KUKA KRL program: ItemPick.src, ItemPick.dat

--- ItemPick.src ---
&ACCESS RVP
&PARAM EDITMASK = *
DEF ItemPick()
   ; ItemPickExample
   ; --------------
   ; Demonstrates bin-picking using roboception's ItemPick module with continuous detection
   ; and pick-and-place operations.
   ;
   ; The program:
   ; 1. Continuously detects items in a bin using vision system
   ; 2. For each detected item, attempts multiple grasp poses if needed
   ; 3. Places successfully picked items at a predefined location
   ; 4. Loops until no more items are detected or program is interrupted
   ;
   ; ENHANCEMENTS:
   ; - Clean 3-tier speed hierarchy (High/Medium/Slow) for easy configuration
   ; - Collision detection support with gripper ID and pre-grasp offsets
   ; - Proper separation of movement offsets vs. detection offsets
   ; - Consistent use of .dat file variables for better maintainability
   ;

   ; Parameters for detection - declared in .dat file
   DECL INT CURRENTITEM, IT

   ; Service name - same as the EKI service name
   ; TODO: Change this to the correct service name - could be "sensor_a_pipeline_1_rc_itempick-compute_grasps"
   serviceNameDetect[] = "rc_itempick-compute_grasps"

   ; Maximum number of grasps to process per detection
   MAX_GRASPS_TO_PROCESS = 1
   ; Maximum number of detection retries
   MAX_DETECTION_RETRIES = 5

   ; Detection parameters
   SUCTION_LENGTH = 0.09  ; Updated to match EKI specification
   SUCTION_WIDTH = 0.02   ; Matches EKI specification
   ITEM_TYPE[] = "BAG"  ; "BAG" for bags or " " for any other item
   LOAD_CARRIER_ID[] = " " ; Single space to represent empty/none
   ROI_ID[] = "roi_bags"
   POSE_FRAME[] = "external"

   ; Collision detection parameters - use " " to skip sending
   GRIPPER_ID[] = "SingleVacuum"    ; Gripper identifier for collision detection
   DET_PRE_GRASP_X_OFFSET = 0.0     ; Detection pre-grasp offset in X direction (m) - SEPARATE from movement offset
   DET_PRE_GRASP_Y_OFFSET = 0.0     ; Detection pre-grasp offset in Y direction (m) - SEPARATE from movement offset
   DET_PRE_GRASP_Z_OFFSET = -0.1    ; Detection pre-grasp offset in Z direction (m) - SEPARATE from movement offset

   ; Gripping parameters
   PRE_GRASP_Z_OFFSET = -100   ; in 100 mm above (along item frame z)
   PRE_PLACE_Z_OFFSET = -100   ; in mm (along world z)

   ; NOTE: Movement uses PRE_GRASP_Z_OFFSET, detection uses DET_PRE_GRASP_Z_OFFSET
   ; These are two different parameters that can be configured independently!

   ;FOLD INI;%{PE}
      ;FOLD BASISTECH INI
         GLOBAL INTERRUPT DECL 3 WHEN $STOPMESS==TRUE DO IR_STOPM ( )
         INTERRUPT ON 3
         BAS (#INITMOV,0 )
      ;ENDFOLD (BASISTECH INI)
   ;ENDFOLD (INI)

   INTERRUPT DECL 89 WHEN $flag[998] DO RC_NOTIFYRECEIVED(1, 998)
   INTERRUPT ON 89

   ;FOLD SPTP home vel=75 % HIGH Speed Transit ;%{pe}
      SPTP XHOME WITH $VEL_AXIS[1] = SVEL_JOINT(ptpSpeedHigh)
   ;ENDFOLD

   GRIPPERBLOW()

   RC_INIT(serviceNameDetect[])

   ;
   ; Main program loop
   ; Continuously tries to detect and pick items until no more items are found
   ; or the program is interrupted
   ;
   LOOP
      RC_SETMSG("Detect next item.")

      ;
      ; Detection retry loop
      ; Attempts to detect items up to MAX_DETECTION_RETRIES times
      ; Exits either on successful detection or when max retries are reached
      ;
      FOR IT = 1 TO MAX_DETECTION_RETRIES
         ; Configure detection parameters using helper function
         ; Sets up item type, pose frame, load carrier, ROI, suction surface, and collision detection parameters
         RC_CONFIGUREPARAMS(serviceNameDetect[], ITEM_TYPE[], POSE_FRAME[], LOAD_CARRIER_ID[], ROI_ID[], SUCTION_LENGTH, SUCTION_WIDTH, GRIPPER_ID[], DET_PRE_GRASP_X_OFFSET, DET_PRE_GRASP_Y_OFFSET, DET_PRE_GRASP_Z_OFFSET)

         ; Perform detection
         ; Sends detection request to vision system and waits for response
         PerformDetection(serviceNameDetect[])

         ; Exit retry loop if detection was successful
         IF DetectionSuccessful() THEN
            EXIT
         ENDIF

         ; Exit program if we've exhausted all retries
         IF IT == MAX_DETECTION_RETRIES THEN
            RC_SETMSG("No more items detected - ending program")
            EXIT
         ENDIF
      ENDFOR

      ;
      ; Process detected grasps
      ; If detection was successful, attempt to pick and place each detected grasp
      ; If detection failed, exit the program
      ;
      IF DetectionSuccessful() THEN
         ; Process grasps from this detection, up to MAX_GRASPS_TO_PROCESS
         FOR CURRENTITEM = 1 TO NUMDETECTEDGRASPS
            GRASP = DETECTEDGRASPS[CURRENTITEM]
            LogGraspInfo(CURRENTITEM, GRASP)
            ExecutePickAndPlace(GRASP, PLACEPOSE, PRE_GRASP_Z_OFFSET, PRE_PLACE_Z_OFFSET)

            ; Break if we've processed maximum number of grasps
            IF CURRENTITEM >= MAX_GRASPS_TO_PROCESS THEN
               EXIT
            ENDIF
         ENDFOR
      ELSE
         ; No items detected after all retries - exit program
         EXIT
      ENDIF
   ENDLOOP

   ; Clean up and return home

   ;FOLD SPTP home vel=75 % HIGH Speed Transit ;%{pe}
      SPTP XHOME WITH $VEL_AXIS[1] = SVEL_JOINT(ptpSpeedHigh)
   ;ENDFOLD
END

DEF ExecutePickAndPlace(GRASPPOSE:IN, PLACEPOSE:IN, PRE_GRASP_Z_OFFSET:IN, PRE_PLACE_Z_OFFSET:IN)
   ;
   ; Executes a complete pick and place operation
   ;
   ; @param GRASPPOSE: Target pose for grasping the object
   ; @param PLACEPOSE: Target pose for placing the object
   ; @param PRE_GRASP_Z_OFFSET: Vertical offset (mm) for pre-grasp approach position
   ; @param PRE_PLACE_Z_OFFSET: Vertical offset (mm) for pre-place approach position
   ; @return TRUE if operation successful, FALSE if vacuum check fails
   ;
   DECL FRAME GRASPPOSE
   DECL E6POS PLACEPOSE
   DECL REAL PRE_GRASP_Z_OFFSET, PRE_PLACE_Z_OFFSET

   ; Internal pose calculations
   DECL FRAME PREGRASPPOSE, PREPLACEPOSE
   DECL FRAME F_OFFSET

   ; Calculate pre-grasp pose
   F_OFFSET = $NULLFRAME
   F_OFFSET.Z = PRE_GRASP_Z_OFFSET
   PREGRASPPOSE = GRASPPOSE:F_OFFSET

   ; Calculate pre-place pose
   PREPLACEPOSE.x = PLACEPOSE.x
   PREPLACEPOSE.y = PLACEPOSE.y
   PREPLACEPOSE.z = PLACEPOSE.z - PRE_PLACE_Z_OFFSET
   PREPLACEPOSE.a = PLACEPOSE.a
   PREPLACEPOSE.b = PLACEPOSE.b
   PREPLACEPOSE.c = PLACEPOSE.c

   ; Move over bin - HIGH speed transit
   SPTP OVERBINPOSE WITH $VEL_AXIS[1] = SVEL_JOINT(ptpSpeedHigh)

   ; Move to pre-grasp - MEDIUM speed approach
   SLIN PREGRASPPOSE with $vel = svel_cp(linSpeedMedium, , lDatMedium), $tool = stool2(fDatDefault), $base = sbase(fDatDefault.base_no)

   ; Move to grasp - SLOW speed for careful in-bin movement
   SLIN GRASPPOSE with $vel = svel_cp(linSpeedSlow, , lDatSlow), $tool = stool2(fDatDefault), $base = sbase(fDatDefault.base_no)

   RC_SETMSG("Grasp position reached. Suctioning...")
   GRIPPERSUCK()

   ; Exit bin - SLOW speed for careful movement out of bin
   SLIN PREGRASPPOSE with $vel = svel_cp(linSpeedSlow, , lDatSlow), $tool = stool2(fDatDefault), $base = sbase(fDatDefault.base_no)

   IF GripperHasVacuumIO THEN
      ; Execute place sequence - HIGH speed transit to place area
      SPTP PREPLACEPOSE with $vel_axis[1] = svel_joint(ptpSpeedHigh), $tool = stool2(fDatDefault), $base = sbase(fDatDefault.base_no), $ipo_mode = sipo_mode(fDatDefault.ipo_frame), $load = sload(fDatDefault.tool_no), $acc_axis[1] = sacc_joint(pDatHigh), $apo = SAPO_PTP(pDatHigh), $gear_jerk[1] = sgear_jerk(pDatHigh), $collmon_tol_pro[1] = use_cm_pro_values(0)
      ; Place item - MEDIUM speed for controlled placement
      SLIN PLACEPOSE with $vel = svel_cp(linSpeedMedium, , lDatMedium), $tool = stool2(fDatDefault), $base = sbase(fDatDefault.base_no)
      GRIPPERBLOW()
      ; Return from place - HIGH speed transit movement
      SPTP PREPLACEPOSE with $vel_axis[1] = svel_joint(ptpSpeedHigh), $tool = stool2(fDatDefault), $base = sbase(fDatDefault.base_no), $ipo_mode = sipo_mode(fDatDefault.ipo_frame), $load = sload(fDatDefault.tool_no), $acc_axis[1] = sacc_joint(pDatHigh), $apo = SAPO_PTP(pDatHigh), $gear_jerk[1] = sgear_jerk(pDatHigh), $collmon_tol_pro[1] = use_cm_pro_values(0)
   ELSE
      RC_SETMSG("No vacuum - moving on...")
      GRIPPERBLOW()
   ENDIF
END

; ---- Helper Functions ----
;FOLD GRIPPERSUCK
   DEF GRIPPERSUCK()
      WAIT SEC 0.0
      GripperBlowIO = false
      GripperSuckIO = true
      WAIT SEC 1.0
   END
;ENDFOLD (GRIPPERSUCK)

;FOLD GRIPPERBLOW
   DEF GRIPPERBLOW()
      WAIT SEC 0.0
      GripperBlowIO = true
      GripperSuckIO = false
   END
;ENDFOLD (GRIPPERSUCK)

; ---- Roboception Functions ----
;FOLD ROBOCEPTION_FUNCTIONS
   ;FOLD RC_CONFIGUREPARAMS
      DEF RC_CONFIGUREPARAMS(serviceNameDetect[]:IN, ITEM_TYPE[]:IN, POSE_FRAME[]:IN, LOAD_CARRIER_ID[]:IN, ROI_ID[]:IN, SUCTION_LENGTH:IN, SUCTION_WIDTH:IN, GRIPPER_ID[]:IN, DET_PRE_GRASP_X_OFFSET:IN, DET_PRE_GRASP_Y_OFFSET:IN, DET_PRE_GRASP_Z_OFFSET:IN)
         DECL CHAR serviceNameDetect[]
         DECL CHAR ITEM_TYPE[]
         DECL CHAR POSE_FRAME[]
         DECL CHAR LOAD_CARRIER_ID[]
         DECL CHAR ROI_ID[]
         DECL CHAR GRIPPER_ID[]
         DECL REAL SUCTION_LENGTH, SUCTION_WIDTH
         DECL REAL DET_PRE_GRASP_X_OFFSET, DET_PRE_GRASP_Y_OFFSET, DET_PRE_GRASP_Z_OFFSET
         DECL EKI_STATUS RET
         DECL E6POS flangePose

         flangePose = $POS_ACT_MES : INV_POS($TOOL)

         ; Core detection parameters
         RET = EKI_SETREAL(serviceNameDetect[], "req/args/suction_surface_length", SUCTION_LENGTH)
         RET = EKI_SETREAL(serviceNameDetect[], "req/args/suction_surface_width", SUCTION_WIDTH)
         RET = EKI_SETSTRING(serviceNameDetect[], "req/args/pose_frame", POSE_FRAME[])
         RET = EKI_SETFRAME(serviceNameDetect[], "req/args/robot_pose", flangePose)

         ; Conditional parameters - send only if not empty
         IF ITEM_TYPE[1] <> " " THEN
            RET = EKI_SETSTRING(serviceNameDetect[], "req/args/item_models/le/type", ITEM_TYPE[])
         ENDIF

         IF ROI_ID[1] <> " " THEN
            RET = EKI_SETSTRING(serviceNameDetect[], "req/args/region_of_interest_id", ROI_ID[])
         ENDIF

         IF LOAD_CARRIER_ID[1] <> " " THEN
            RET = EKI_SETSTRING(serviceNameDetect[], "req/args/load_carrier_id", LOAD_CARRIER_ID[])
         ENDIF

         IF GRIPPER_ID[1] <> " " THEN
            RET = EKI_SetString(serviceNameDetect[], "req/args/collision_detection/@gripper_id", GRIPPER_ID[])
         ENDIF

         IF DET_PRE_GRASP_X_OFFSET <> 0.0 THEN
            RET = EKI_SetReal(serviceNameDetect[], "req/args/collision_detection/pre_grasp_offset/@x", DET_PRE_GRASP_X_OFFSET)
         ENDIF

         IF DET_PRE_GRASP_Y_OFFSET <> 0.0 THEN
            RET = EKI_SetReal(serviceNameDetect[], "req/args/collision_detection/pre_grasp_offset/@y", DET_PRE_GRASP_Y_OFFSET)
         ENDIF

         IF DET_PRE_GRASP_Z_OFFSET <> 0.0 THEN
            RET = EKI_SetReal(serviceNameDetect[], "req/args/collision_detection/pre_grasp_offset/@z", DET_PRE_GRASP_Z_OFFSET)
         ENDIF
      END
   ;ENDFOLD (RC_CONFIGUREPARAMS)

   ;FOLD RC_SETMSG
      DEF RC_SETMSG(msg[]:IN)
         DECL CHAR msg[]
         DECL KrlMsgPar_T PARAMS[3]
         RC_SETMSG_PARAM(msg[], PARAMS[])
      END
   ;ENDFOLD (RC_SETMSG)

   ;FOLD RC_SETMSG_PARAM
      DEF RC_SETMSG_PARAM(msg[]:IN, PARAMS:OUT)
         DECL CHAR msg[]
         DECL KrlMsgPar_T PARAMS[]

         DECL KrlMsg_T name
         DECL KrlMsgOpt_T options
         DECL INT handle, len, count
         DECL EKrlMsgType type

         name={modul[] "rc", nr 1, msg_txt[] " "}

         type=#notify

         len=STRLEN(msg[])
         IF len>0 THEN
            IF len>80 THEN
               len=80
            ENDIF
            FOR count=1 TO len
               name.msg_txt[count]=msg[count]
            ENDFOR
         ELSE
            name.msg_txt[]="parameter msg[] is missing"
         ENDIF

         handle=Set_KrlMsg(type, name, PARAMS[], options)
      END
   ;ENDFOLD (RC_SETMSG_PARAM)

   ;FOLD RC_INIT
      DEF RC_INIT(configfilename[]:IN)
         DECL CHAR configfilename[]
         DECL EKI_STATUS RET
         RET = EKI_INIT(configfilename[])
      END
   ;ENDFOLD (RC_INIT)

   ;FOLD RC_OPENCONNECTION
      DEF RC_OPENCONNECTION(configfilename[]:IN)
         DECL CHAR configfilename[]
         DECL EKI_STATUS RET
         RET = EKI_Open(configfilename[])
         EKI_CHECK(RET,#Quit)
      END
   ;ENDFOLD (RC_OPENCONNECTION)

   ;FOLD RC_CLOSECONNECTION
      DEF RC_CLOSECONNECTION(configfilename[]:IN, strplace[]:IN)
         DECL CHAR configfilename[]
         DECL CHAR strplace[]
         DECL EKI_STATUS RET
         WAIT SEC 0
         RET = EKI_Close(configfilename[])
         RET = EKI_ClearBuffer(configfilename[], strplace[])
      END
   ;ENDFOLD (RC_CLOSECONNECTION)

   ;FOLD RC_WAITFORRESULT
      DEF RC_WAITFORRESULT(waitflag:IN)
         DECL INT waitflag

         WAIT FOR $FLAG[waitflag] OR NOT $FLAG[RCEkiAliveFlagNo]

         ; EKI-connection has been closed
         IF(NOT $FLAG[RCEkiAliveFlagNo]) THEN
            RC_SETMSG("EKI connection lost")
         ENDIF

         $FLAG[waitflag] = FALSE
         WAIT SEC 0
      END
   ;ENDFOLD (RC_WAITFORRESULT)

   ;FOLD RC_NOTIFYRECEIVED
      DEF RC_NOTIFYRECEIVED(waitflag:IN, eofresulflag:IN)
         DECL INT waitflag
         DECL INT eofresulflag
         $FLAG[eofresulflag]=FALSE
         $FLAG[waitflag]=TRUE
      END
   ;ENDFOLD (RC_NOTIFYRECEIVED)

   ;FOLD RC_READRESULT
      DEF RC_READRESULT(configFileName[]:IN)
         DECL CHAR configFileName[]
         DECL RETURNCODE_T RESULT
         DECL EKI_STATUS RET
         DECL INT j
         DECL FRAME POSE
         DECL KrlMsgPar_T par[3]

         POSE = POSE_IDENT

         RESULT={VALUE 0, MSG[] "0"}

         RET = EKI_GetInt(configFileName[], "res/return_code/@value", RESULT.VALUE)
         RET = EKI_GetString(configFileName[], "res/return_code/@message", RESULT.MSG[])
         RETURNCODE = RESULT

         ; Display error message immediately if there is one
         IF (RESULT.VALUE < 0) THEN
            RC_SETMSG("API Error")
            RC_SETMSG(RESULT.MSG[])
         ENDIF

         RET = EKI_CheckBuffer(configFileName[], "res/grasps/le/uuid")
         NUMDETECTEDGRASPS = RET.Buff

         ; Log the number of detected grasps
         par[1] = {par_type #value, par_INT 0}
         par[1].par_INT = NUMDETECTEDGRASPS
         RC_SETMSG_PARAM("Number of detected grasps: %1", par[])

         ; Only try to get frames if grasps were detected
         IF NUMDETECTEDGRASPS > 0 THEN
            FOR j=1 TO NUMDETECTEDGRASPS
               RET = EKI_GetFrame(configFileName[], "res/grasps/le/pose", POSE)
               DETECTEDGRASPS[j] = POSE
            ENDFOR
         ELSE
            RC_SETMSG("No grasps detected - skipping pose extraction")
         ENDIF

         RET = EKI_ClearBuffer(configFileName[], "res")
      END
   ;ENDFOLD (RC_READRESULT)

   DEFFCT BOOL DetectionSuccessful()
      IF (RETURNCODE.VALUE < 0) THEN
         RETURN FALSE
      ENDIF

      IF NUMDETECTEDGRASPS > 0 THEN
         RETURN TRUE
      ENDIF

      RETURN FALSE
   ENDFCT

   DEF PerformDetection(serviceNameDetect[]:IN)
      DECL CHAR serviceNameDetect[]
      DECL EKI_Status RET

      ; Open connection before sending request
      RC_OPENCONNECTION(serviceNameDetect[])

      ; Synchronize advance run pointer
      WAIT SEC 0

      ; Send request
      RET = EKI_Send(serviceNameDetect[], "req")

      ; Wait for response and read results
      RC_WAITFORRESULT(1)
      RC_READRESULT(serviceNameDetect[])

      ; Close the connection after reading results
      RC_CLOSECONNECTION(serviceNameDetect[], "req")
   END

   DEF LogGraspInfo(currentGrasp:IN, pose:IN)
      DECL INT currentGrasp
      DECL FRAME pose
      DECL krlmsgpar_t par[4]

      ; Set up parameters for translation message
      par[1] = {par_type #value, par_INT 0}
      par[1].par_INT = currentGrasp
      par[2] = {par_type #value, par_REAL 0}
      par[2].par_REAL = pose.x
      par[3] = {par_type #value, par_REAL 0}
      par[3].par_REAL = pose.y
      par[4] = {par_type #value, par_REAL 0}
      par[4].par_REAL = pose.z

      RC_SETMSG_PARAM("Processing grasp %1: trans: x: %2, y: %3, z: %4", par[])

   END
;ENDFOLD (ROBOCEPTION_FUNCTIONS)

--- ItemPick.dat ---
&ACCESS RVP
&PARAM EDITMASK = *
DEFDAT ItemPick
   ;FOLD EXTERNAL DECLARATIONS;%{PE}%MKUKATPBASIS,%CEXT,%VCOMMON,%P
   ;FOLD BASISTECH EXT;%{PE}%MKUKATPBASIS,%CEXT,%VEXT,%P
   EXT BAS (BAS_COMMAND :IN,REAL :IN)
   ;ENDFOLD (BASISTECH EXT)
   ;FOLD USER EXT;%{E}%MKUKATPUSER,%CEXT,%VEXT,%P

   ; EKI Communication
   DECL CHAR serviceNameDetect[64]

   ; Common structures and variables
   DECL INT RCEkiAliveFlagNo=997
   STRUC RETURNCODE_T INT VALUE,CHAR MSG[512]
   DECL RETURNCODE_T RETURNCODE

   ; Frame declarations
   DECL FRAME GRASP
   DECL FRAME DETECTEDGRASPS[32]
   DECL FRAME POSE_IDENT={X 0.0,Y 0.0,Z 0.0,A 0.0,B 0.0,C 0.0}

   ; IO Signals
   SIGNAL GripperSuckIO $OUT[1]
   SIGNAL GripperBlowIO $OUT[2]
   SIGNAL GripperHasVacuumIO $IN[1]

   ; Detection results
   DECL INT NUMDETECTEDGRASPS

   ; Detection parameters
   DECL CHAR ITEM_TYPE[32]
   DECL CHAR POSE_FRAME[32]
   DECL CHAR LOAD_CARRIER_ID[32]
   DECL CHAR ROI_ID[32]
   DECL CHAR GRIPPER_ID[32]
   DECL REAL SUCTION_LENGTH, SUCTION_WIDTH
   DECL REAL DET_PRE_GRASP_X_OFFSET, DET_PRE_GRASP_Y_OFFSET, DET_PRE_GRASP_Z_OFFSET
   DECL INT MAX_DETECTION_RETRIES
   DECL INT MAX_GRASPS_TO_PROCESS
   DECL EKI_STATUS RET

   ; ==============================================================================
   ; SPEED HIERARCHY - Clean 3-tier system for easy configuration
   ; ==============================================================================

   ; PTP (Joint) Speeds - in percentage
   DECL REAL ptpSpeedHigh=75.0        ; % - Fast transit movements (home, over bin, etc.)
   DECL REAL ptpSpeedMedium=50.0      ; % - Approach movements (to pre-grasp area)
   DECL REAL ptpSpeedSlow=25.0        ; % - Careful movements near workpiece

   ; Linear (Cartesian) Speeds - in m/s
   DECL REAL linSpeedHigh=0.400       ; m/s - Fast linear movements (over bin, transit)
   DECL REAL linSpeedMedium=0.200     ; m/s - Approach movements (to pre-grasp)
   DECL REAL linSpeedSlow=0.080       ; m/s - Careful in-bin operations

   ; Legacy speeds - DEPRECATED (kept for compatibility)
   DECL REAL rlinVelocityStd=0.25    ; m/s
   DECL REAL rlinVelocitySlow=0.15   ; m/s
   DECL REAL rptpVelocityStd=10      ; %

   ; Movement parameter offsets
   DECL REAL PRE_GRASP_Z_OFFSET         ; in mm
   DECL REAL PRE_PLACE_Z_OFFSET

   ; Positions
   DECL E6POS XHOME={X 212.898911,Y -2.87642241,Z 569.476624,A -90.000,B 0.0,C -180.000,S 2,T 2,E1 0.0,E2 0.0,E3 0.0,E4 0.0,E5 0.0,E6 0.0}
   DECL E6POS OVERBINPOSE={X -18.2943077,Y 621.050415,Z 246.103409,A -80.0664063,B 0.0205745194,C -179.997696,S 2,T 11,E1 0.0,E2 0.0,E3 0.0,E4 0.0,E5 0.0,E6 0.0}
   DECL E6POS PLACEPOSE={X 565.796,Y -85,Z -60,A 0,B 0,C -180,S 2,T 35,E1 0.0,E2 0.0,E3 0.0,E4 0.0,E5 0.0,E6 0.0}

   ; ==============================================================================
   ; MOVEMENT DATA STRUCTURES - Consistent speed configurations
   ; ==============================================================================

   ; Linear movement data structures - Clean 3-tier system
   DECL LDAT lDatHigh={VEL 0.400,ACC 20.0000,APO_DIST 10.0000,APO_FAC 50.0000,AXIS_VEL 100.000,AXIS_ACC 100.000,ORI_TYP #VAR,CIRC_TYP #BASE,JERK_FAC 50.0000,GEAR_JERK 100.000,EXAX_IGN 0,CB {AUX_PT {ORI #CONSIDER,E1 #CONSIDER,E2 #CONSIDER,E3 #CONSIDER,E4 #CONSIDER,E5 #CONSIDER,E6 #CONSIDER},TARGET_PT {ORI #INTERPOLATE,E1 #INTERPOLATE,E2 #INTERPOLATE,E3 #INTERPOLATE,E4 #INTERPOLATE,E5 #INTERPOLATE,E6 #INTERPOLATE}}}

   DECL LDAT lDatMedium={VEL 0.200,ACC 20.0000,APO_DIST 10.0000,APO_FAC 50.0000,AXIS_VEL 100.000,AXIS_ACC 100.000,ORI_TYP #VAR,CIRC_TYP #BASE,JERK_FAC 50.0000,GEAR_JERK 100.000,EXAX_IGN 0,CB {AUX_PT {ORI #CONSIDER,E1 #CONSIDER,E2 #CONSIDER,E3 #CONSIDER,E4 #CONSIDER,E5 #CONSIDER,E6 #CONSIDER},TARGET_PT {ORI #INTERPOLATE,E1 #INTERPOLATE,E2 #INTERPOLATE,E3 #INTERPOLATE,E4 #INTERPOLATE,E5 #INTERPOLATE,E6 #INTERPOLATE}}}

   DECL LDAT lDatSlow={VEL 0.080,ACC 20.0000,APO_DIST 10.0000,APO_FAC 50.0000,AXIS_VEL 100.000,AXIS_ACC 100.000,ORI_TYP #VAR,CIRC_TYP #BASE,JERK_FAC 50.0000,GEAR_JERK 100.000,EXAX_IGN 0,CB {AUX_PT {ORI #CONSIDER,E1 #CONSIDER,E2 #CONSIDER,E3 #CONSIDER,E4 #CONSIDER,E5 #CONSIDER,E6 #CONSIDER},TARGET_PT {ORI #INTERPOLATE,E1 #INTERPOLATE,E2 #INTERPOLATE,E3 #INTERPOLATE,E4 #INTERPOLATE,E5 #INTERPOLATE,E6 #INTERPOLATE}}}

   ; PTP movement data structures - Clean 3-tier system
   DECL PDAT pDatHigh={VEL 75.0000,ACC 20.0000,APO_DIST 50.0000,APO_MODE #CDIS,GEAR_JERK 100.000,EXAX_IGN 0}
   DECL PDAT pDatMedium={VEL 50.0000,ACC 20.0000,APO_DIST 30.0000,APO_MODE #CDIS,GEAR_JERK 100.000,EXAX_IGN 0}
   DECL PDAT pDatSlow={VEL 25.0000,ACC 20.0000,APO_DIST 10.0000,APO_MODE #CDIS,GEAR_JERK 100.000,EXAX_IGN 0}

   ; Frame data (unchanged)
   DECL FDAT fDatDefault={TOOL_NO 4,BASE_NO 0,IPO_FRAME #BASE,POINT2[] " "}

   ; Legacy movement data - DEPRECATED (kept for compatibility)
   DECL LDAT lDatDefault={VEL 2.00000,ACC 20.0000,APO_DIST 10.0000,APO_FAC 50.0000,AXIS_VEL 100.000,AXIS_ACC 100.000,ORI_TYP #VAR,CIRC_TYP #BASE,JERK_FAC 50.0000,GEAR_JERK 100.000,EXAX_IGN 0,CB {AUX_PT {ORI #CONSIDER,E1 #CONSIDER,E2 #CONSIDER,E3 #CONSIDER,E4 #CONSIDER,E5 #CONSIDER,E6 #CONSIDER},TARGET_PT {ORI #INTERPOLATE,E1 #INTERPOLATE,E2 #INTERPOLATE,E3 #INTERPOLATE,E4 #INTERPOLATE,E5 #INTERPOLATE,E6 #INTERPOLATE}}}
   DECL PDAT pDatDefault={VEL 10.0000,ACC 20.0000,APO_DIST 10.0000,APO_MODE #CDIS,GEAR_JERK 100.000,EXAX_IGN 0}

   ; ==============================================================================
   ; COLLISION DETECTION PARAMETERS - declared above with detection parameters
   ; ==============================================================================
   ; These are user-configurable parameters that can be set at the top of the program
   ; Use " " (single space) to skip sending a parameter
   ; GRIPPER_ID and DET_PRE_GRASP_*_OFFSET are already declared above

   ;ENDFOLD (USER EXT)
   ;ENDFOLD (EXTERNAL DECLARATIONS)
ENDDAT
